Yaskawa INFORM job: P_X_MP.JBI

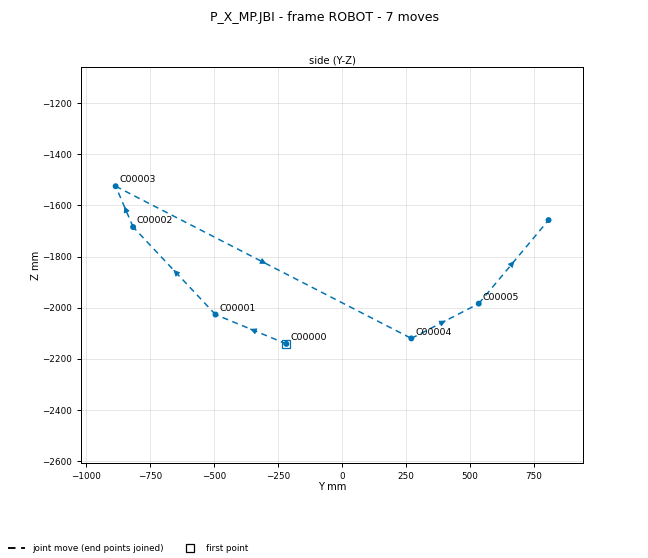
[picture p0: tool path of P_X_MP.JBI in frame ROBOT, 7 of 7 moves have a stored position in this frame; points joined in program order, loops and branches not executed]
/JOB
//NAME P_X_MP
///FOLDERNAME INNE
//POS
///NPOS 7,7,7,0,0,0
///TOOL 0
///POSTYPE ROBOT
///RECTAN
///RCONF 0,0,0,0,0,0,0,0,0,0,0,0,0,0,0,0,0,0,0,0,0,0,0,0
C00000=1028.869,-218.314,-2141.103,-0.0032,0.0034,-90.0044
C00001=1028.242,-495.272,-2026.450,0.0010,-20.5455,-90.0095
C00002=1027.339,-817.296,-1684.302,0.0077,-47.4931,-90.0141
C00003=1027.088,-885.729,-1524.739,0.0079,-47.4935,-90.0158
C00004=1029.488,270.579,-2119.775,-0.0092,30.5462,-90.0102
C00005=1029.960,534.219,-1983.759,-0.0148,50.0873,-90.0131
C00006=1030.505,807.199,-1657.102,-0.0759,76.8689,-90.0777
BC00000=650.660,6920.928,1262.163
BC00001=650.660,6920.928,1262.163
BC00002=650.660,6920.928,1262.163
BC00003=650.660,6920.928,1262.163
BC00004=650.660,6920.928,1262.163
BC00005=650.660,6920.928,1262.163
BC00006=650.660,6920.928,1262.163
///POSTYPE PULSE
///PULSE
EC00000=0,0
EC00001=-167491,0
EC00002=-431280,0
EC00003=-525386,0
EC00004=274969,0
EC00005=440232,0
EC00006=678625,0
//INST
///DATE 2023/10/04 15:13
///ATTR SC,RW,RJ
////FRAME ROBOT
///GROUP1 RB1,BS1
///GROUP2 ST1
NOP
MOVJ C00000 BC00000 VJ=0.78  +MOVJ EC00000 VJ=0.78
MOVJ C00001 BC00001 VJ=0.78  +MOVJ EC00001 VJ=0.78
MOVJ C00002 BC00002 VJ=0.78  +MOVJ EC00002 VJ=0.78
MOVJ C00003 BC00003 VJ=0.78  +MOVJ EC00003 VJ=0.78
MOVJ C00004 BC00004 VJ=0.78  +MOVJ EC00004 VJ=0.78
MOVJ C00005 BC00005 VJ=0.78  +MOVJ EC00005 VJ=0.78
MOVJ C00006 BC00006 VJ=0.78  +MOVJ EC00006 VJ=0.78
END
